PROGRAM P_KNX_Communication
VAR
	KL6301_0: KL6301;
	
	bActivate             : BOOL := TRUE;
	idx                   : INT := 1;
	EIB_PHYS_ADDR         : EIB_PHYS_ADDR := (Area := 1, Line := 6, Device := 150);
	EIB_GROUP_FILTER      : ARRAY [1..8] OF EIB_GROUP_FILTER := [(
																	GROUP_ADDR := (MAIN := 12, SUB_MAIN := 0, NUMBER := 0),
																	GROUP_LEN  := 63
																)];
	iMode                 : INT := 0;
	tTimeout              : TIME := T#5S;
	
	bActive               : BOOL;
	bReady                : BOOL;
	bError                : BOOL;
	iErrorId              : EIB_Error_Code;
	
END_VAR

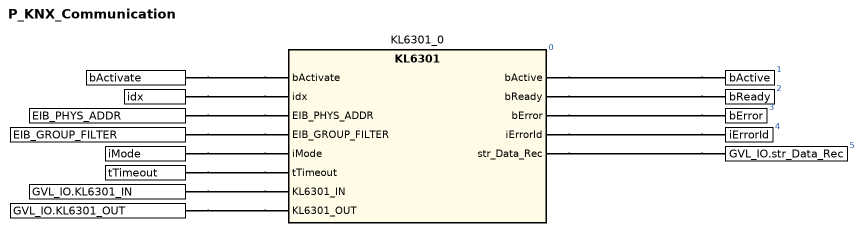
KL6301_0(
    bActivate := bActivate,
    idx := idx,
    EIB_PHYS_ADDR := EIB_PHYS_ADDR,
    EIB_GROUP_FILTER := EIB_GROUP_FILTER,
    iMode := iMode,
    tTimeout := tTimeout,
    KL6301_IN := GVL_IO.KL6301_IN,
    KL6301_OUT := GVL_IO.KL6301_OUT); // KL6301
bActive := KL6301_0.bActive;
bReady := KL6301_0.bReady;
bError := KL6301_0.bError;
iErrorId := KL6301_0.iErrorId;
GVL_IO.str_Data_Rec := KL6301_0.str_Data_Rec;

END_PROGRAM

(* stored: Version 1.1.0.1, ProductVersion 3.1.4024.5
   POU P_KNX_Communication: Id {02b5d330-ac60-478d-9585-2c0731be3ad1}, SpecialFunc None *)
